INTERFACE I_Subject

METHOD Attach
VAR_INPUT
	ipObserver	: I_Observer;
END_VAR
END_METHOD

METHOD Detach
VAR_INPUT
END_VAR
END_METHOD

END_INTERFACE

(* stored: Version 1.1.0.1, ProductVersion 3.1.4024.9
   Itf I_Subject: Id {f7ca362b-2d38-4db5-9e26-173f77c8712d}
   Method Attach: Id {c9c8f916-2283-45d3-83cd-a6a37f088420}
   Method Detach: Id {5f9884af-b656-49c0-982a-734534651c4a} *)
